# EPICS autosave request: iocBoot/ioc13InstekGPP_1/auto_settings.req
file InstekGPP_settings.req    P=$(P), R=$(R)"
file pid_control_settings.req  P=$(P), PID=PID1
file pid_control_settings.req  P=$(P), PID=PID2
